// Mitsubishi GX Works2 project: 10   PLC: FX3U/FX3UC

PROGRAM MAIN
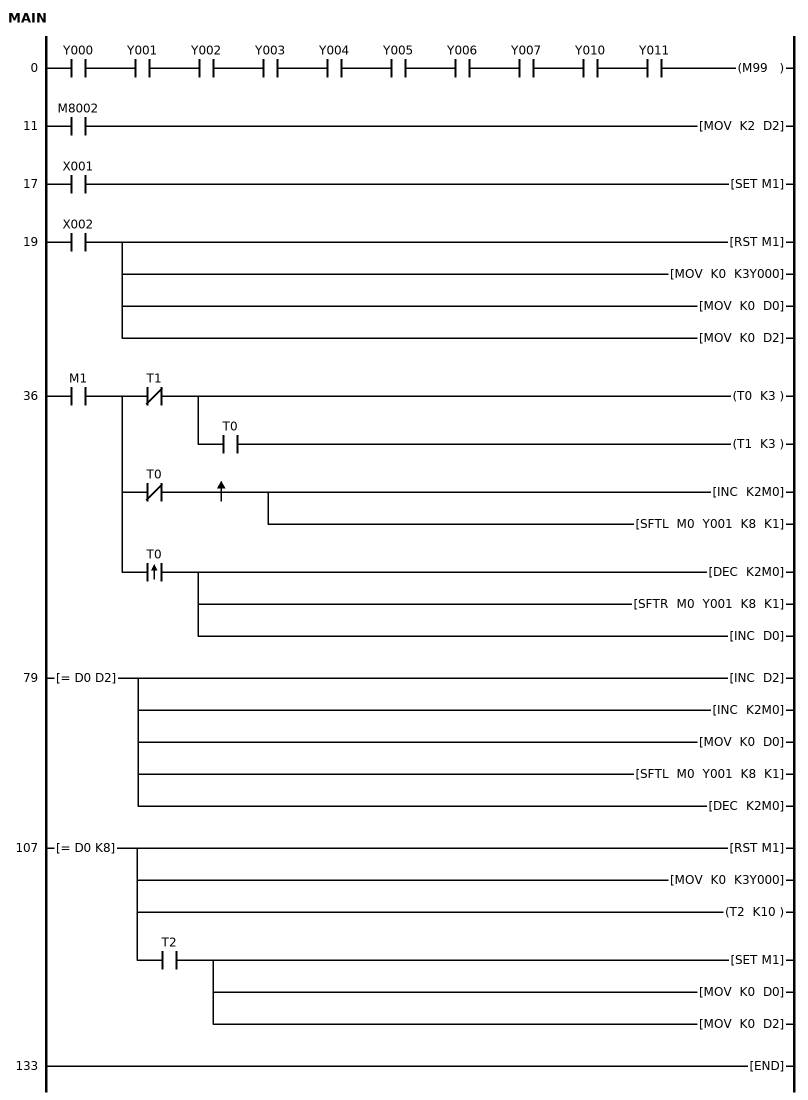
0     LD      Y000
      AND     Y001
      AND     Y002
      AND     Y003
      AND     Y004
      AND     Y005
      AND     Y006
      AND     Y007
      AND     Y010
      AND     Y011
      OUT     M99
11    LD      M8002
      MOV     K2 D2
17    LD      X001
      SET     M1
19    LD      X002
      RST     M1
      MOV     K0 K3Y000
      MOV     K0 D0
      MOV     K0 D2
36    LD      M1
      MPS
      ANI     T1
      OUT     T0 K3
      AND     T0
      OUT     T1 K3
      MRD
      ANI     T0
      MEP
      INC     K2M0
      SFTL    M0 Y001 K8 K1
      MPP
      ANDP    T0
      DEC     K2M0
      SFTR    M0 Y001 K8 K1
      INC     D0
79    LD=     D0 D2
      INC     D2
      INC     K2M0
      MOV     K0 D0
      SFTL    M0 Y001 K8 K1
      DEC     K2M0
107   LD=     D0 K8
      RST     M1
      MOV     K0 K3Y000
      OUT     T2 K10
      AND     T2
      SET     M1
      MOV     K0 D0
      MOV     K0 D2
133   END
END_PROGRAM
